(* Logix 5000 project; controller SX_V040001_C001 vendor 1 type 14 code 77 rev 16.22; software revision 16.04; part 11 of 35 *)
(* tags used below, declared in another part *)
   ALL_KINDS : INT[90];
   Basic : INT;
   DRIVE : INT[32];
   DRIVE_INTERVAL : INT[8];
   EMPTYING : INT[18];
   G_AOutput : DINT[8];
   G_DInput : DINT[3];
   G_DOutput : DINT[3];
   METERING : INT[44];
   METERING_PULSE : DINT[14];
   negi_param398 : DINT;
   PARAMETER : INT[501];
   T_ACT_DATA_RESET : TIMER;
   T_CHOCO_PRESS_LOW : TIMER;
   T_DEL_DATA : TIMER;
   T_OUTLET_CLOSE : TIMER;
   T_RUN_OUT_CHOCOPUMP : TIMER;
(* MainProgram, continued *)

ROUTINE Emptying   (* ladder *)
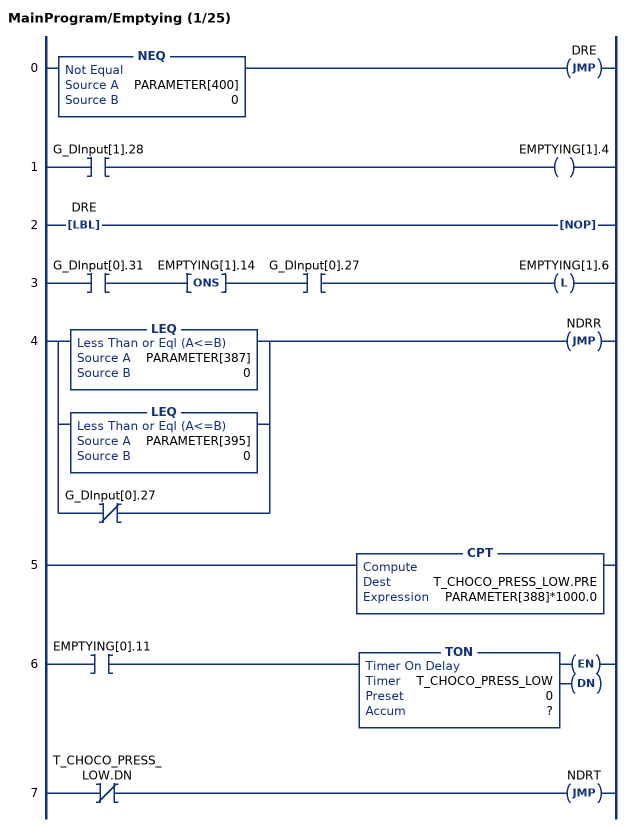
   0: NEQ(PARAMETER[400],0)JMP(DRE);
   1: XIC(G_DInput[1].28)OTE(EMPTYING[1].4);
   2: LBL(DRE)NOP();
   3: XIC(G_DInput[0].31)ONS(EMPTYING[1].14)XIC(G_DInput[0].27)OTL(EMPTYING[1].6);
   4: [LEQ(PARAMETER[387],0) ,LEQ(PARAMETER[395],0) ,XIO(G_DInput[0].27) ]JMP(NDRR);
   5: CPT(T_CHOCO_PRESS_LOW.PRE,PARAMETER[388]*1000.0);
   6: XIC(EMPTYING[0].11)TON(T_CHOCO_PRESS_LOW,?,?);
   7: XIO(T_CHOCO_PRESS_LOW.DN)JMP(NDRT);
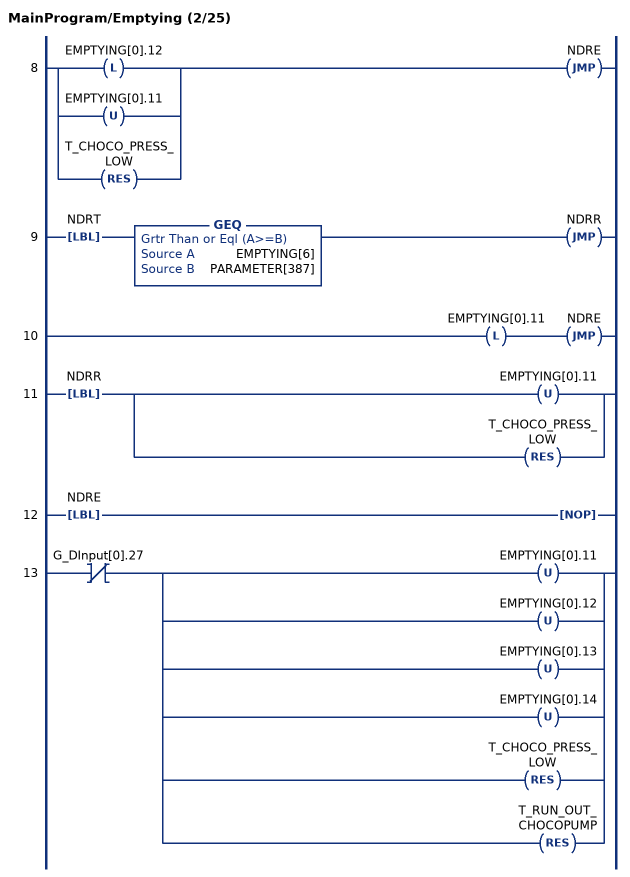
   8: [OTL(EMPTYING[0].12) ,OTU(EMPTYING[0].11) ,RES(T_CHOCO_PRESS_LOW) ]JMP(NDRE);
   9: LBL(NDRT)GEQ(EMPTYING[6],PARAMETER[387])JMP(NDRR);
   10: OTL(EMPTYING[0].11)JMP(NDRE);
   11: LBL(NDRR)[OTU(EMPTYING[0].11) ,RES(T_CHOCO_PRESS_LOW) ];
   12: LBL(NDRE)NOP();
   13: XIO(G_DInput[0].27)[OTU(EMPTYING[0].11) ,OTU(EMPTYING[0].12) ,OTU(EMPTYING[0].13) ,OTU(EMPTYING[0].14) ,RES(T_CHOCO_PRESS_LOW) ,RES(T_RUN_OUT_CHOCOPUMP) ];
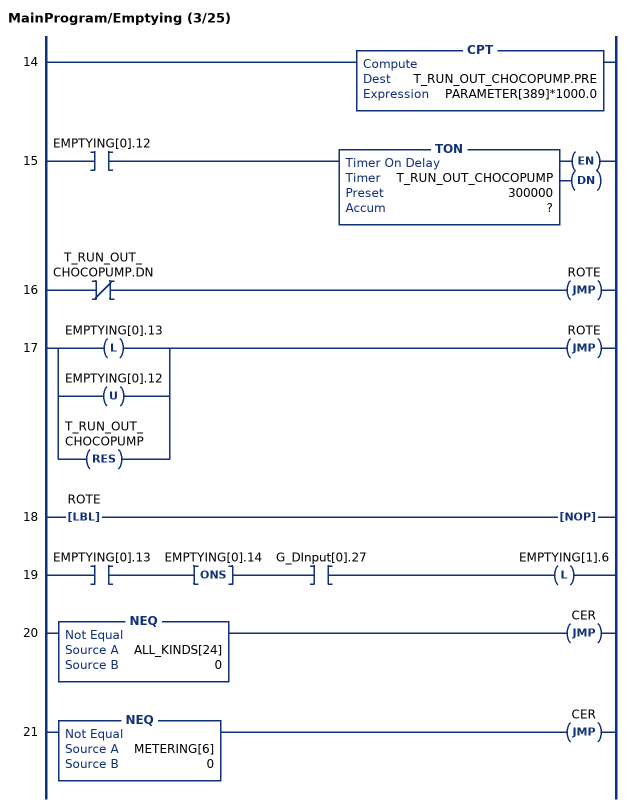
   14: CPT(T_RUN_OUT_CHOCOPUMP.PRE,PARAMETER[389]*1000.0);
   15: XIC(EMPTYING[0].12)TON(T_RUN_OUT_CHOCOPUMP,?,?);
   16: XIO(T_RUN_OUT_CHOCOPUMP.DN)JMP(ROTE);
   17: [OTL(EMPTYING[0].13) ,OTU(EMPTYING[0].12) ,RES(T_RUN_OUT_CHOCOPUMP) ]JMP(ROTE);
   18: LBL(ROTE)NOP();
   19: XIC(EMPTYING[0].13)ONS(EMPTYING[0].14)XIC(G_DInput[0].27)OTL(EMPTYING[1].6);
   20: NEQ(ALL_KINDS[24],0)JMP(CER);
   21: NEQ(METERING[6],0)JMP(CER);
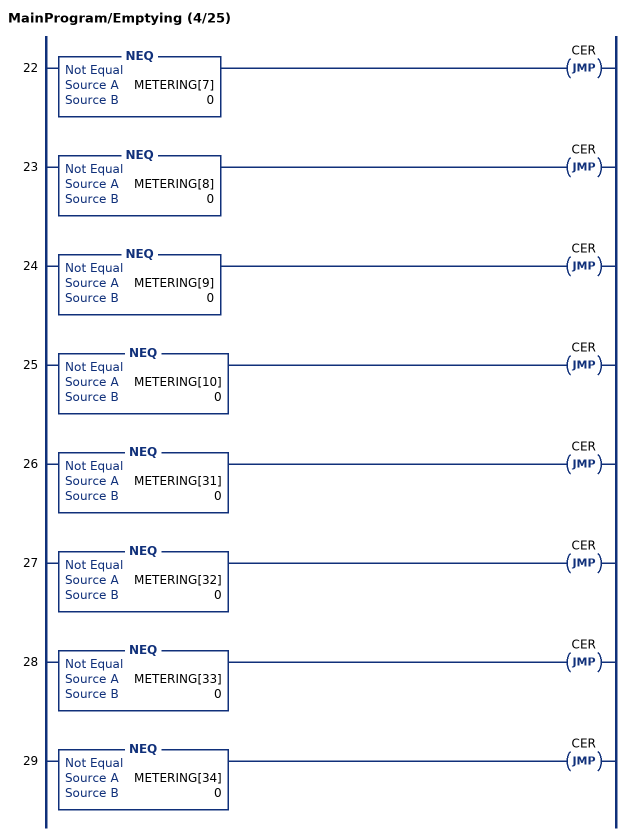
   22: NEQ(METERING[7],0)JMP(CER);
   23: NEQ(METERING[8],0)JMP(CER);
   24: NEQ(METERING[9],0)JMP(CER);
   25: NEQ(METERING[10],0)JMP(CER);
   26: NEQ(METERING[31],0)JMP(CER);
   27: NEQ(METERING[32],0)JMP(CER);
   28: NEQ(METERING[33],0)JMP(CER);
   29: NEQ(METERING[34],0)JMP(CER);
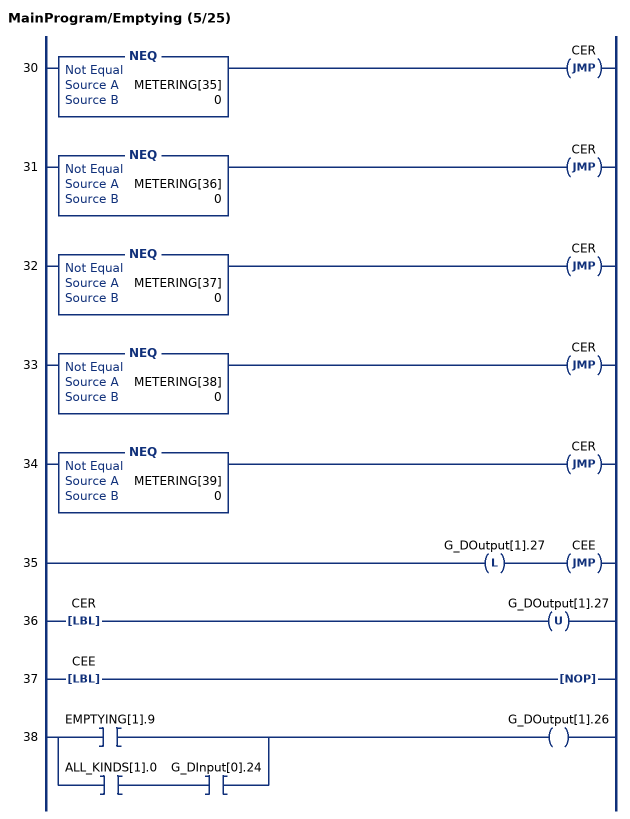
   30: NEQ(METERING[35],0)JMP(CER);
   31: NEQ(METERING[36],0)JMP(CER);
   32: NEQ(METERING[37],0)JMP(CER);
   33: NEQ(METERING[38],0)JMP(CER);
   34: NEQ(METERING[39],0)JMP(CER);
   35: OTL(G_DOutput[1].27)JMP(CEE);
   36: LBL(CER)OTU(G_DOutput[1].27);
   37: LBL(CEE)NOP();
   38: [XIC(EMPTYING[1].9) ,XIC(ALL_KINDS[1].0) XIC(G_DInput[0].24) ]OTE(G_DOutput[1].26);
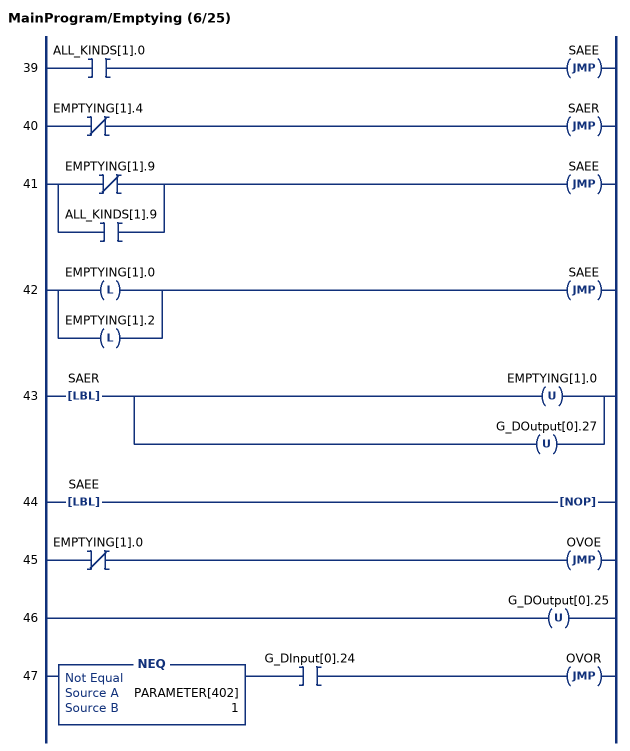
   39: XIC(ALL_KINDS[1].0)JMP(SAEE);
   40: XIO(EMPTYING[1].4)JMP(SAER);
   41: [XIO(EMPTYING[1].9) ,XIC(ALL_KINDS[1].9) ]JMP(SAEE);
   42: [OTL(EMPTYING[1].0) ,OTL(EMPTYING[1].2) ]JMP(SAEE);
   43: LBL(SAER)[OTU(EMPTYING[1].0) ,OTU(G_DOutput[0].27) ];
   44: LBL(SAEE)NOP();
   45: XIO(EMPTYING[1].0)JMP(OVOE);
   46: OTU(G_DOutput[0].25);
   47: NEQ(PARAMETER[402],1)XIC(G_DInput[0].24)JMP(OVOR);
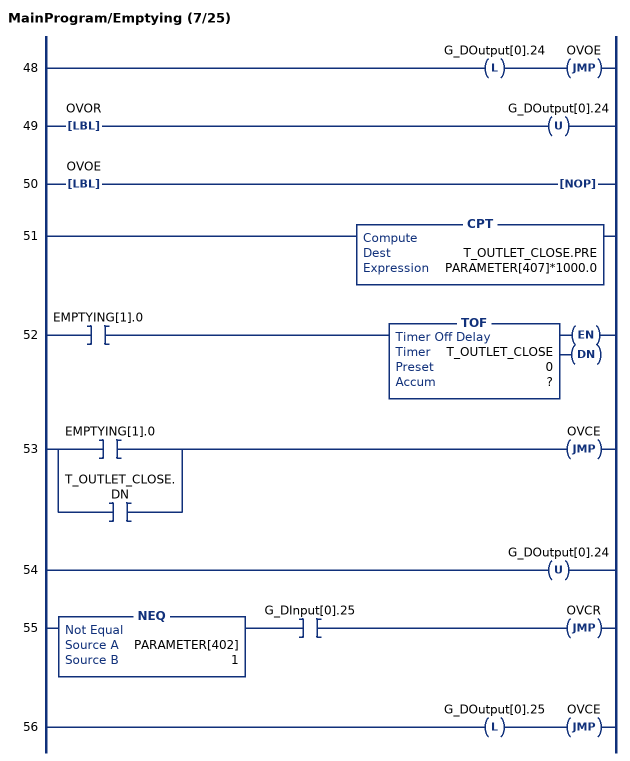
   48: OTL(G_DOutput[0].24)JMP(OVOE);
   49: LBL(OVOR)OTU(G_DOutput[0].24);
   50: LBL(OVOE)NOP();
   51: CPT(T_OUTLET_CLOSE.PRE,PARAMETER[407]*1000.0);
   52: XIC(EMPTYING[1].0)TOF(T_OUTLET_CLOSE,?,?);
   53: [XIC(EMPTYING[1].0) ,XIC(T_OUTLET_CLOSE.DN) ]JMP(OVCE);
   54: OTU(G_DOutput[0].24);
   55: NEQ(PARAMETER[402],1)XIC(G_DInput[0].25)JMP(OVCR);
   56: OTL(G_DOutput[0].25)JMP(OVCE);
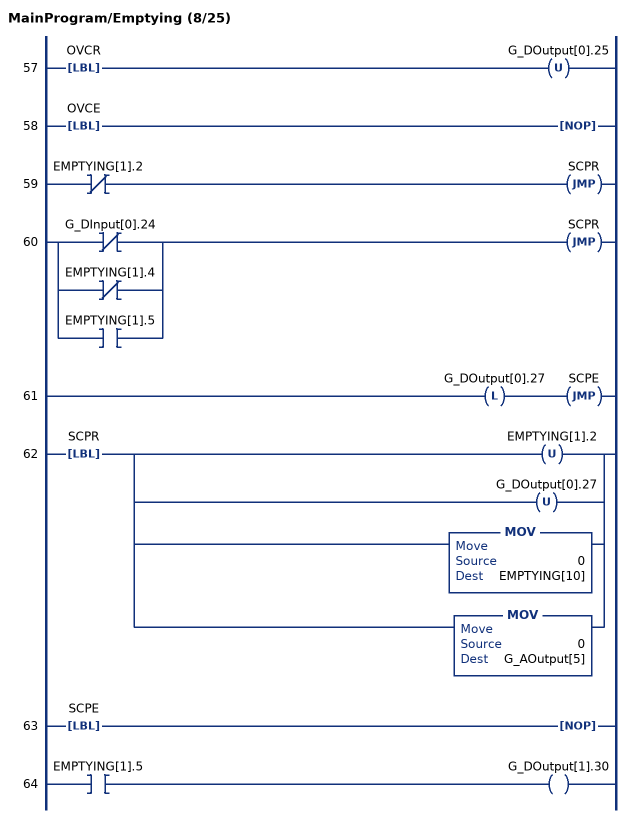
   57: LBL(OVCR)OTU(G_DOutput[0].25);
   58: LBL(OVCE)NOP();
   59: XIO(EMPTYING[1].2)JMP(SCPR);
   60: [XIO(G_DInput[0].24) ,XIO(EMPTYING[1].4) ,XIC(EMPTYING[1].5) ]JMP(SCPR);
   61: OTL(G_DOutput[0].27)JMP(SCPE);
   62: LBL(SCPR)[OTU(EMPTYING[1].2) ,OTU(G_DOutput[0].27) ,MOV(0,EMPTYING[10]) ,MOV(0,G_AOutput[5]) ];
   63: LBL(SCPE)NOP();
   64: XIC(EMPTYING[1].5)OTE(G_DOutput[1].30);
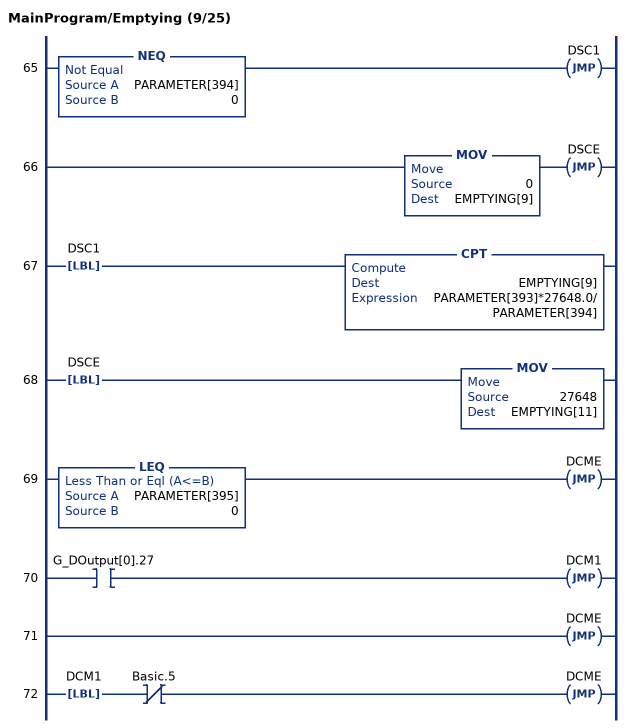
   65: NEQ(PARAMETER[394],0)JMP(DSC1);
   66: MOV(0,EMPTYING[9])JMP(DSCE);
   67: LBL(DSC1)CPT(EMPTYING[9],PARAMETER[393]*27648.0/PARAMETER[394]);
   68: LBL(DSCE)MOV(27648,EMPTYING[11]);
   69: LEQ(PARAMETER[395],0)JMP(DCME);
   70: XIC(G_DOutput[0].27)JMP(DCM1);
   71: JMP(DCME);
   72: LBL(DCM1)XIO(Basic.5)JMP(DCME);
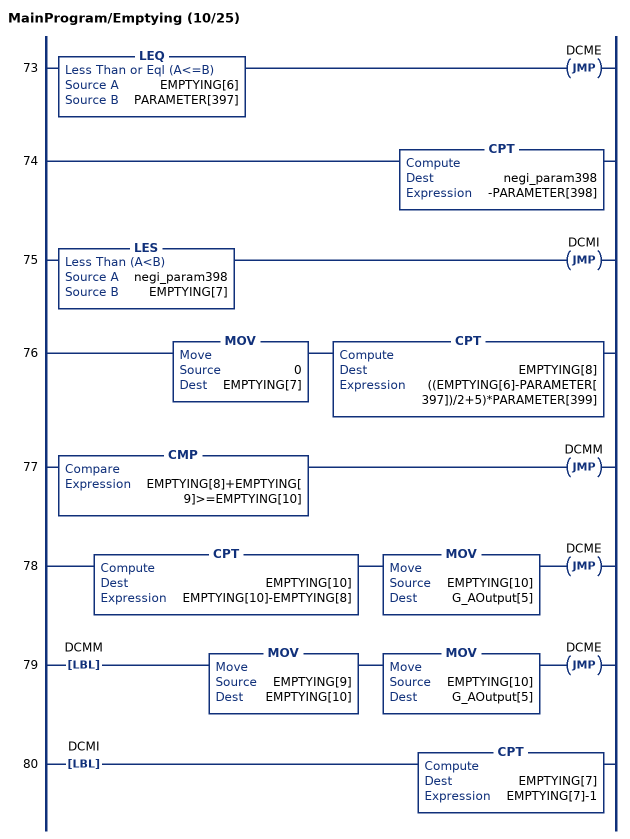
   73: LEQ(EMPTYING[6],PARAMETER[397])JMP(DCME);
   74: CPT(negi_param398,-PARAMETER[398]);
   75: LES(negi_param398,EMPTYING[7])JMP(DCMI);
   76: MOV(0,EMPTYING[7])CPT(EMPTYING[8],((EMPTYING[6]-PARAMETER[397])/2+5)*PARAMETER[399]);
   77: CMP(EMPTYING[8]+EMPTYING[9]>=EMPTYING[10])JMP(DCMM);
   78: CPT(EMPTYING[10],EMPTYING[10]-EMPTYING[8])MOV(EMPTYING[10],G_AOutput[5])JMP(DCME);
   79: LBL(DCMM)MOV(EMPTYING[9],EMPTYING[10])MOV(EMPTYING[10],G_AOutput[5])JMP(DCME);
   80: LBL(DCMI)CPT(EMPTYING[7],EMPTYING[7]-1);
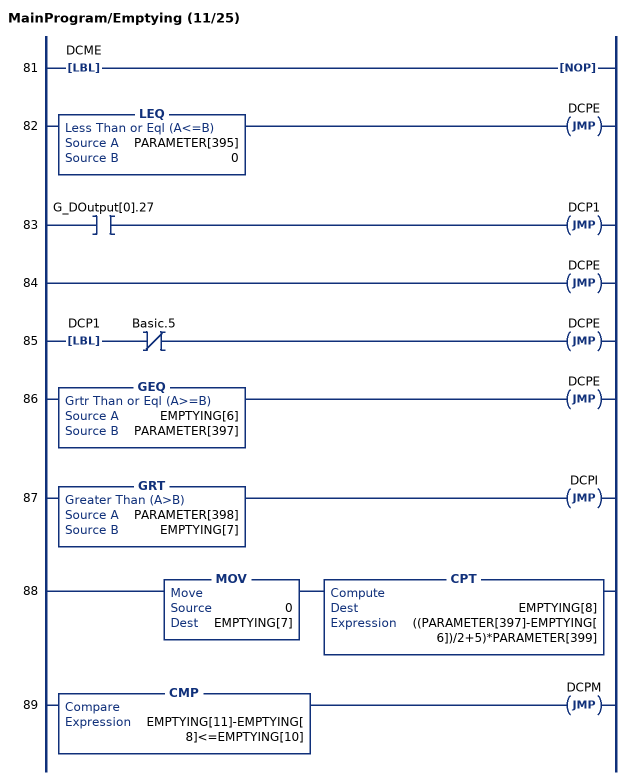
   81: LBL(DCME)NOP();
   82: LEQ(PARAMETER[395],0)JMP(DCPE);
   83: XIC(G_DOutput[0].27)JMP(DCP1);
   84: JMP(DCPE);
   85: LBL(DCP1)XIO(Basic.5)JMP(DCPE);
   86: GEQ(EMPTYING[6],PARAMETER[397])JMP(DCPE);
   87: GRT(PARAMETER[398],EMPTYING[7])JMP(DCPI);
   88: MOV(0,EMPTYING[7])CPT(EMPTYING[8],((PARAMETER[397]-EMPTYING[6])/2+5)*PARAMETER[399]);
   89: CMP(EMPTYING[11]-EMPTYING[8]<=EMPTYING[10])JMP(DCPM);
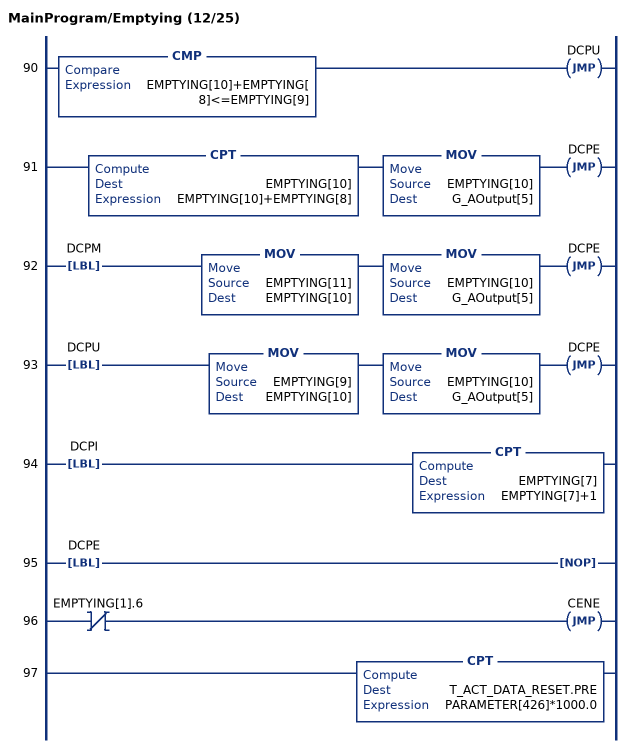
   90: CMP(EMPTYING[10]+EMPTYING[8]<=EMPTYING[9])JMP(DCPU);
   91: CPT(EMPTYING[10],EMPTYING[10]+EMPTYING[8])MOV(EMPTYING[10],G_AOutput[5])JMP(DCPE);
   92: LBL(DCPM)MOV(EMPTYING[11],EMPTYING[10])MOV(EMPTYING[10],G_AOutput[5])JMP(DCPE);
   93: LBL(DCPU)MOV(EMPTYING[9],EMPTYING[10])MOV(EMPTYING[10],G_AOutput[5])JMP(DCPE);
   94: LBL(DCPI)CPT(EMPTYING[7],EMPTYING[7]+1);
   95: LBL(DCPE)NOP();
   96: XIO(EMPTYING[1].6)JMP(CENE);
   97: CPT(T_ACT_DATA_RESET.PRE,PARAMETER[426]*1000.0);
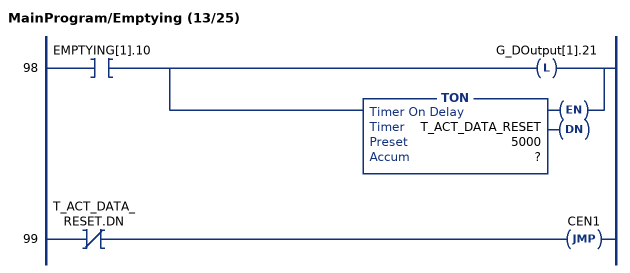
   98: XIC(EMPTYING[1].10)[OTL(G_DOutput[1].21) ,TON(T_ACT_DATA_RESET,?,?) ];
   99: XIO(T_ACT_DATA_RESET.DN)JMP(CEN1);
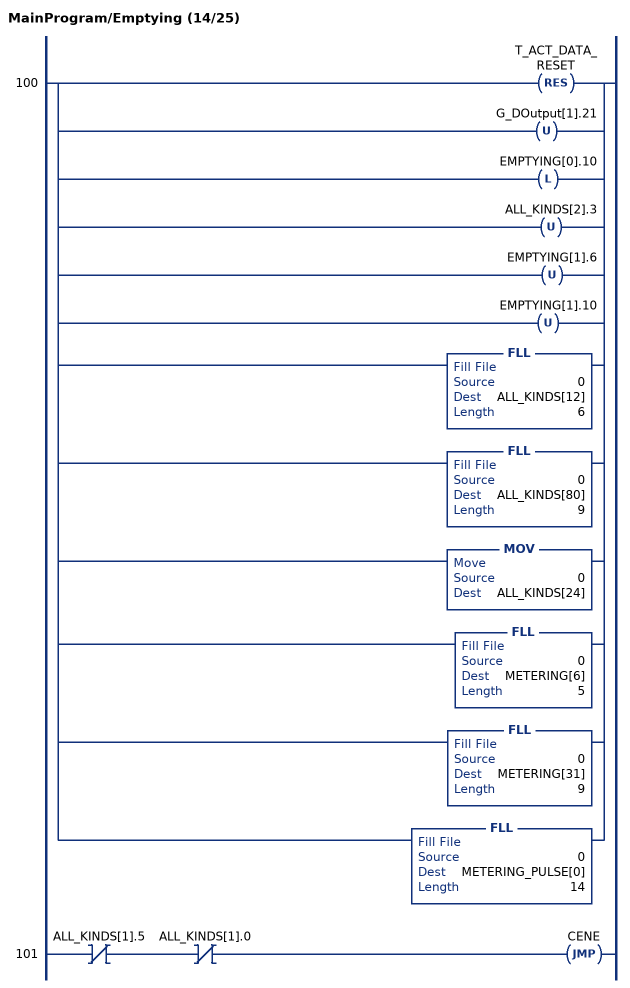
   100: [RES(T_ACT_DATA_RESET) ,OTU(G_DOutput[1].21) ,OTL(EMPTYING[0].10) ,OTU(ALL_KINDS[2].3) ,OTU(EMPTYING[1].6) ,OTU(EMPTYING[1].10) ,FLL(0,ALL_KINDS[12],6) ,FLL(0,ALL_KINDS[80],9) ,MOV(0,ALL_KINDS[24]) ,FLL(0,METERING[6],5) ,FLL(0,METERING[31],9) ,FLL(0,METERING_PULSE[0],14) ];
   101: XIO(ALL_KINDS[1].5)XIO(ALL_KINDS[1].0)JMP(CENE);
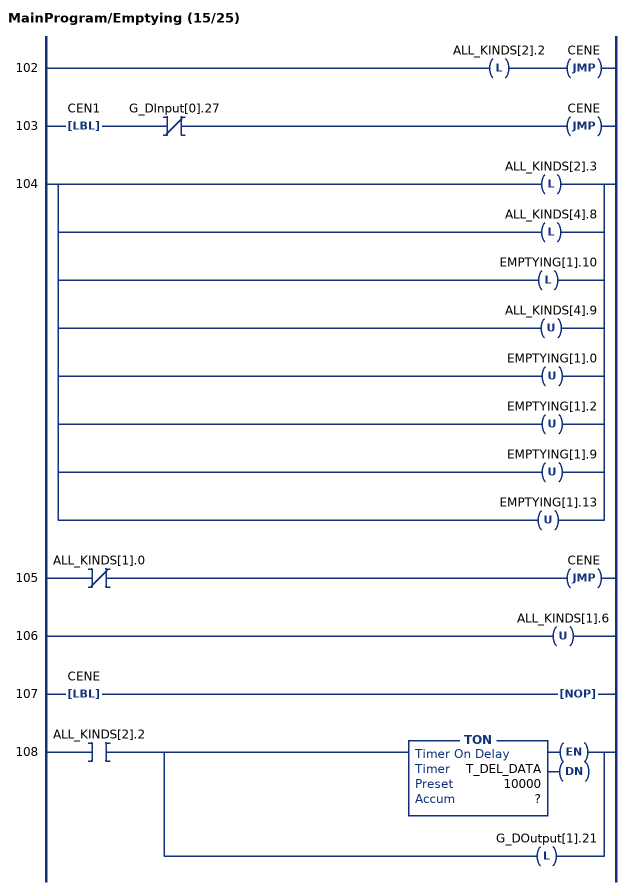
   102: OTL(ALL_KINDS[2].2)JMP(CENE);
   103: LBL(CEN1)XIO(G_DInput[0].27)JMP(CENE);
   104: [OTL(ALL_KINDS[2].3) ,OTL(ALL_KINDS[4].8) ,OTL(EMPTYING[1].10) ,OTU(ALL_KINDS[4].9) ,OTU(EMPTYING[1].0) ,OTU(EMPTYING[1].2) ,OTU(EMPTYING[1].9) ,OTU(EMPTYING[1].13) ];
   105: XIO(ALL_KINDS[1].0)JMP(CENE);
   106: OTU(ALL_KINDS[1].6);
   107: LBL(CENE)NOP();
   108: XIC(ALL_KINDS[2].2)[TON(T_DEL_DATA,?,?) ,OTL(G_DOutput[1].21) ];
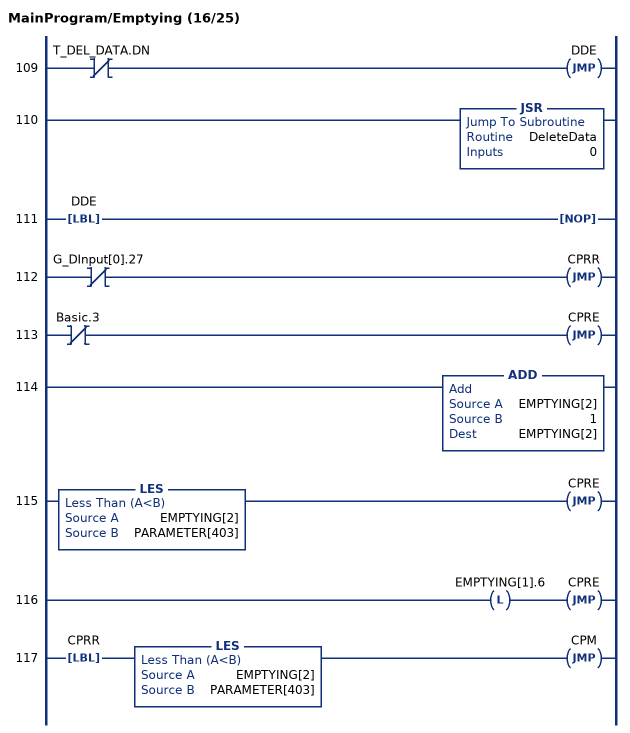
   109: XIO(T_DEL_DATA.DN)JMP(DDE);
   110: JSR(DeleteData,0);
   111: LBL(DDE)NOP();
   112: XIO(G_DInput[0].27)JMP(CPRR);
   113: XIO(Basic.3)JMP(CPRE);
   114: ADD(EMPTYING[2],1,EMPTYING[2]);
   115: LES(EMPTYING[2],PARAMETER[403])JMP(CPRE);
   116: OTL(EMPTYING[1].6)JMP(CPRE);
   117: LBL(CPRR)LES(EMPTYING[2],PARAMETER[403])JMP(CPM);
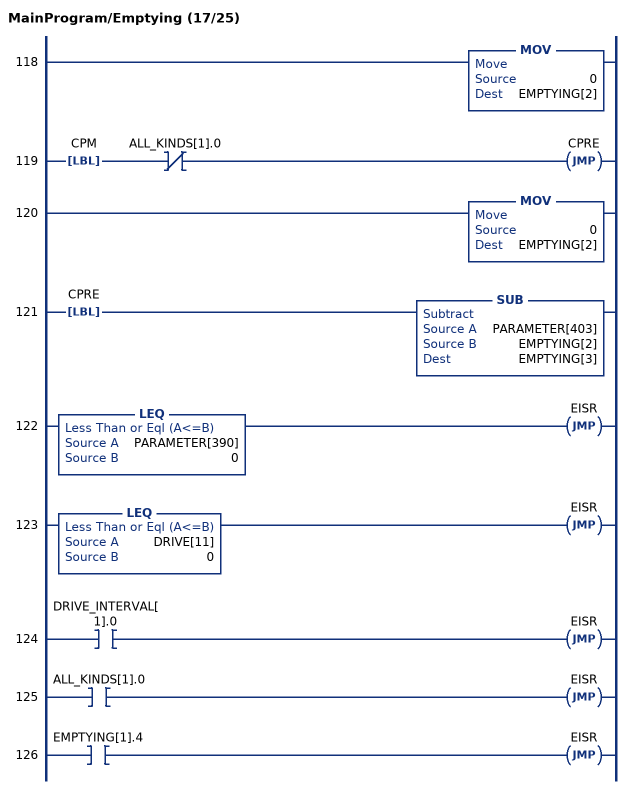
   118: MOV(0,EMPTYING[2]);
   119: LBL(CPM)XIO(ALL_KINDS[1].0)JMP(CPRE);
   120: MOV(0,EMPTYING[2]);
   121: LBL(CPRE)SUB(PARAMETER[403],EMPTYING[2],EMPTYING[3]);
   122: LEQ(PARAMETER[390],0)JMP(EISR);
   123: LEQ(DRIVE[11],0)JMP(EISR);
   124: XIC(DRIVE_INTERVAL[1].0)JMP(EISR);
   125: XIC(ALL_KINDS[1].0)JMP(EISR);
   126: XIC(EMPTYING[1].4)JMP(EISR);
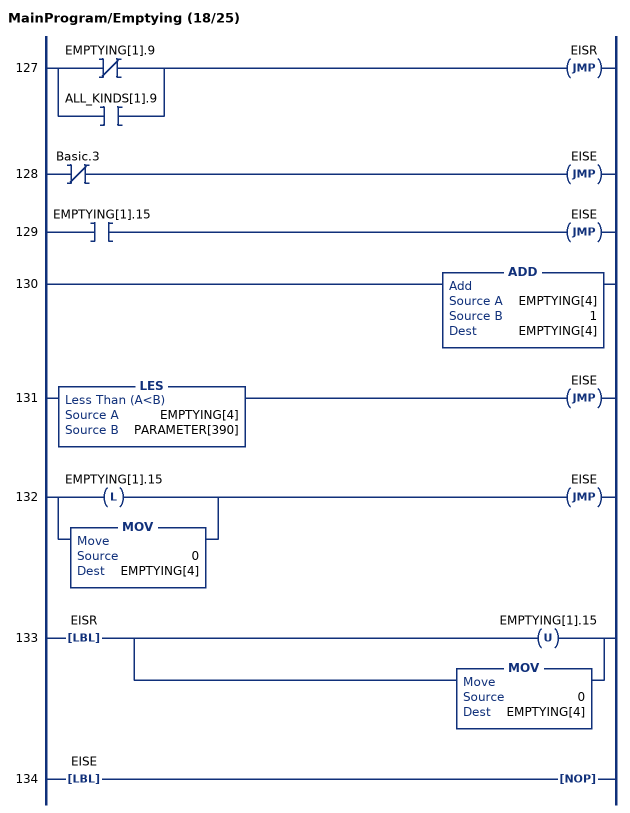
   127: [XIO(EMPTYING[1].9) ,XIC(ALL_KINDS[1].9) ]JMP(EISR);
   128: XIO(Basic.3)JMP(EISE);
   129: XIC(EMPTYING[1].15)JMP(EISE);
   130: ADD(EMPTYING[4],1,EMPTYING[4]);
   131: LES(EMPTYING[4],PARAMETER[390])JMP(EISE);
   132: [OTL(EMPTYING[1].15) ,MOV(0,EMPTYING[4]) ]JMP(EISE);
   133: LBL(EISR)[OTU(EMPTYING[1].15) ,MOV(0,EMPTYING[4]) ];
   134: LBL(EISE)NOP();
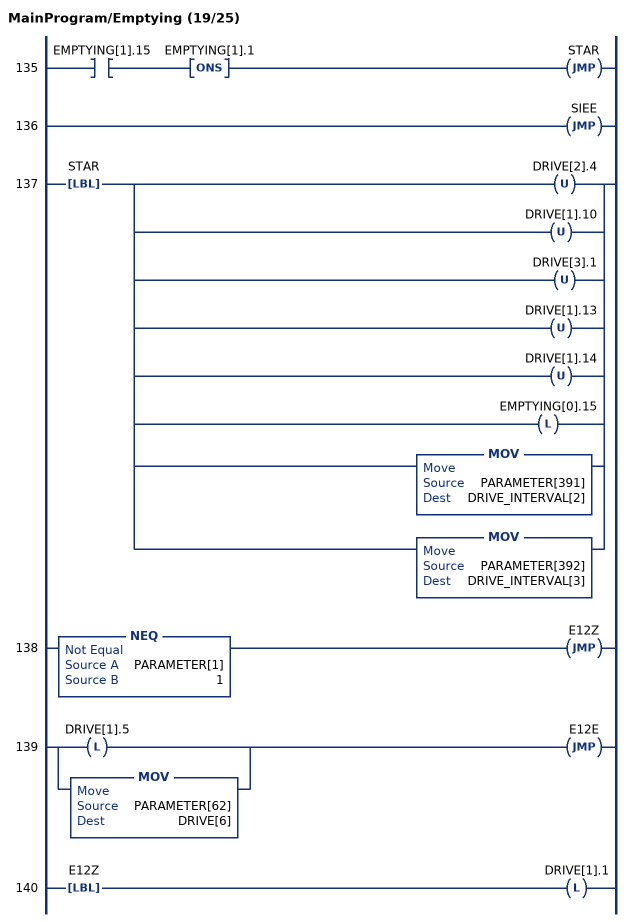
   135: XIC(EMPTYING[1].15)ONS(EMPTYING[1].1)JMP(STAR);
   136: JMP(SIEE);
   137: LBL(STAR)[OTU(DRIVE[2].4) ,OTU(DRIVE[1].10) ,OTU(DRIVE[3].1) ,OTU(DRIVE[1].13) ,OTU(DRIVE[1].14) ,OTL(EMPTYING[0].15) ,MOV(PARAMETER[391],DRIVE_INTERVAL[2]) ,MOV(PARAMETER[392],DRIVE_INTERVAL[3]) ];
   138: NEQ(PARAMETER[1],1)JMP(E12Z);
   139: [OTL(DRIVE[1].5) ,MOV(PARAMETER[62],DRIVE[6]) ]JMP(E12E);
   140: LBL(E12Z)OTL(DRIVE[1].1);
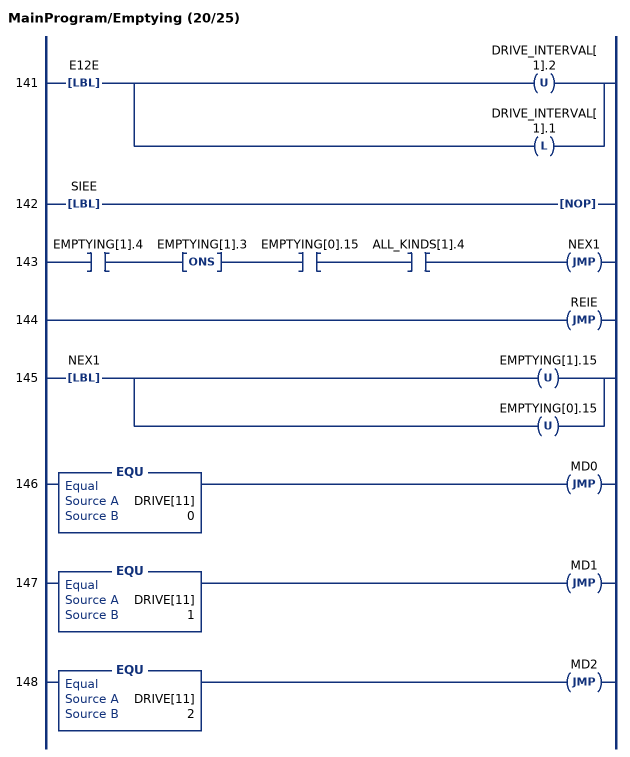
   141: LBL(E12E)[OTU(DRIVE_INTERVAL[1].2) ,OTL(DRIVE_INTERVAL[1].1) ];
   142: LBL(SIEE)NOP();
   143: XIC(EMPTYING[1].4)ONS(EMPTYING[1].3)XIC(EMPTYING[0].15)XIC(ALL_KINDS[1].4)JMP(NEX1);
   144: JMP(REIE);
   145: LBL(NEX1)[OTU(EMPTYING[1].15) ,OTU(EMPTYING[0].15) ];
   146: EQU(DRIVE[11],0)JMP(MD0);
   147: EQU(DRIVE[11],1)JMP(MD1);
   148: EQU(DRIVE[11],2)JMP(MD2);
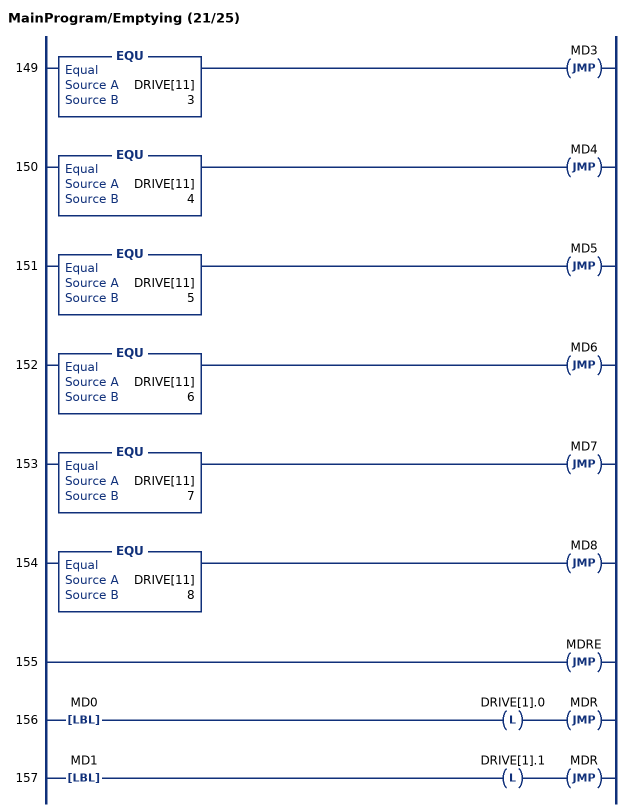
   149: EQU(DRIVE[11],3)JMP(MD3);
   150: EQU(DRIVE[11],4)JMP(MD4);
   151: EQU(DRIVE[11],5)JMP(MD5);
   152: EQU(DRIVE[11],6)JMP(MD6);
   153: EQU(DRIVE[11],7)JMP(MD7);
   154: EQU(DRIVE[11],8)JMP(MD8);
   155: JMP(MDRE);
   156: LBL(MD0)OTL(DRIVE[1].0)JMP(MDR);
   157: LBL(MD1)OTL(DRIVE[1].1)JMP(MDR);
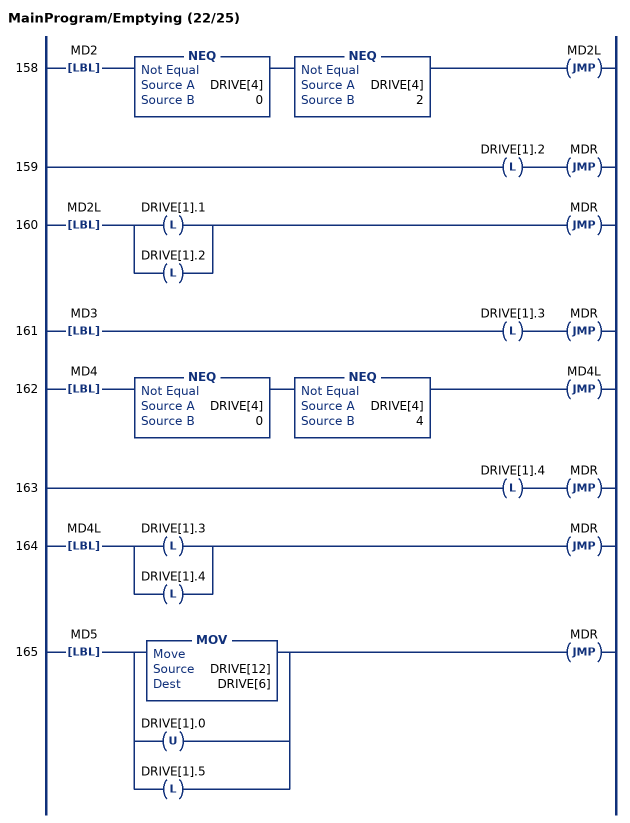
   158: LBL(MD2)NEQ(DRIVE[4],0)NEQ(DRIVE[4],2)JMP(MD2L);
   159: OTL(DRIVE[1].2)JMP(MDR);
   160: LBL(MD2L)[OTL(DRIVE[1].1) ,OTL(DRIVE[1].2) ]JMP(MDR);
   161: LBL(MD3)OTL(DRIVE[1].3)JMP(MDR);
   162: LBL(MD4)NEQ(DRIVE[4],0)NEQ(DRIVE[4],4)JMP(MD4L);
   163: OTL(DRIVE[1].4)JMP(MDR);
   164: LBL(MD4L)[OTL(DRIVE[1].3) ,OTL(DRIVE[1].4) ]JMP(MDR);
   165: LBL(MD5)[MOV(DRIVE[12],DRIVE[6]) ,OTU(DRIVE[1].0) ,OTL(DRIVE[1].5) ]JMP(MDR);
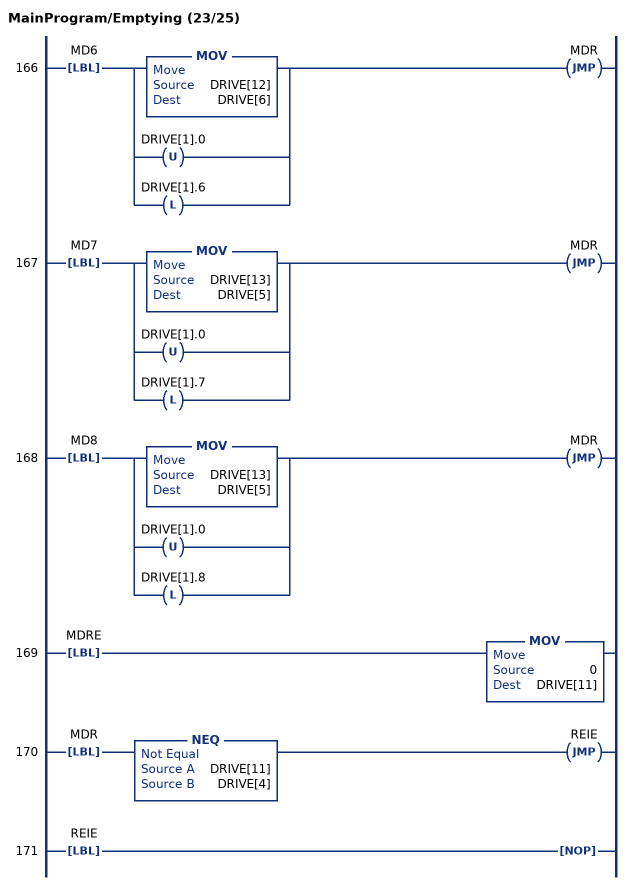
   166: LBL(MD6)[MOV(DRIVE[12],DRIVE[6]) ,OTU(DRIVE[1].0) ,OTL(DRIVE[1].6) ]JMP(MDR);
   167: LBL(MD7)[MOV(DRIVE[13],DRIVE[5]) ,OTU(DRIVE[1].0) ,OTL(DRIVE[1].7) ]JMP(MDR);
   168: LBL(MD8)[MOV(DRIVE[13],DRIVE[5]) ,OTU(DRIVE[1].0) ,OTL(DRIVE[1].8) ]JMP(MDR);
   169: LBL(MDRE)MOV(0,DRIVE[11]);
   170: LBL(MDR)NEQ(DRIVE[11],DRIVE[4])JMP(REIE);
   171: LBL(REIE)NOP();
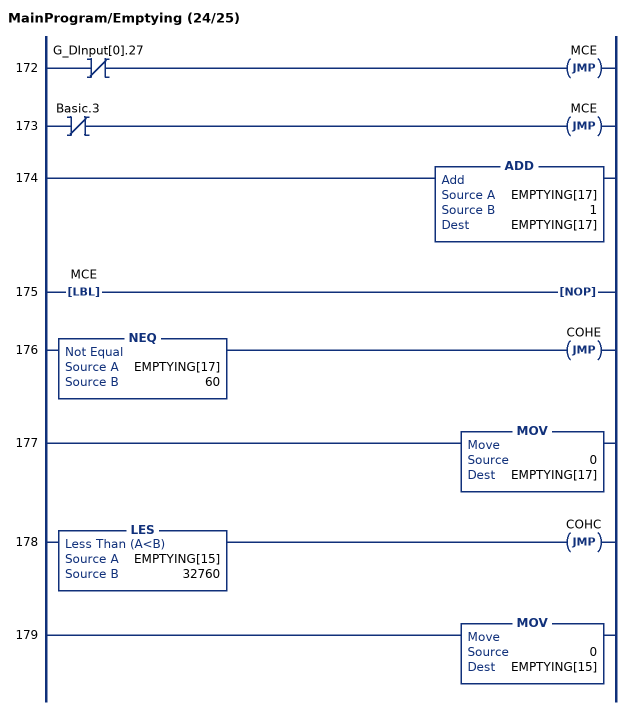
   172: XIO(G_DInput[0].27)JMP(MCE);
   173: XIO(Basic.3)JMP(MCE);
   174: ADD(EMPTYING[17],1,EMPTYING[17]);
   175: LBL(MCE)NOP();
   176: NEQ(EMPTYING[17],60)JMP(COHE);
   177: MOV(0,EMPTYING[17]);
   178: LES(EMPTYING[15],32760)JMP(COHC);
   179: MOV(0,EMPTYING[15]);
